// TIA Portal V19 export
ORGANIZATION_BLOCK "MainBeltLift"   // OB125, FBD, ProgramCycle
TITLE = "Main Program Sweep (Cycle)"
{ S7_Optimized_Access := 'TRUE' }
AUTHOR : Siemens
// Main programm belt lift
// stored: IsIECCheckEnabled true, SetENOAutomatically true
   VAR_INPUT
      Initial_Call : Bool;   // Initial call of this OB
      Remanence : Bool;   // =True, if remanent data are available
   END_VAR
BEGIN

REGION Network 1
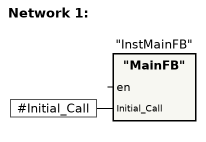
   "InstMainFB"(Initial_Call := #Initial_Call);   // "MainFB"
END_REGION
END_ORGANIZATION_BLOCK
